(* IEC 61131-3 sources: RL_MAR/experiments/comparison/llm4plc/results/gpt-4o_20260507_114630/20260507_122147, 1 file *)

(* ---- generated_code_iteration_0.st ---- *)
plaintext
START_ST
FUNCTION_BLOCK SoilTestingDeviceControl
VAR_INPUT
    StartButton : BOOL; (* Input for starting the testing process *)
    SoilSampleDetected : BOOL; (* Input for detecting soil sample *)
END_VAR
VAR_OUTPUT
    NutrientPump : BOOL; (* Output to control nutrient pump *)
    pHAdjustmentPump : BOOL; (* Output to control pH adjustment pump *)
END_VAR
VAR
    pHSensorValue : REAL; (* Simulated pH sensor value *)
    NutrientSensorValue : REAL; (* Simulated nutrient sensor value *)
    TestingStatus : INT; (* Status: 0=Idle, 1=Testing, 2=Completed *)
    NutrientThreshold : REAL := 0.7; (* Nutrient level threshold for analysis *)
    pHThreshold : REAL := 6.5; (* pH level threshold for analysis *)
END_VAR

(* Function block logic *)
IF TestingStatus = 0 THEN
    (* STATE 0: Idle *)
    NutrientPump := FALSE;
    pHAdjustmentPump := FALSE;
    pHSensorValue := 7.0; (* Initialize pH sensor value *)
    NutrientSensorValue := 0.5; (* Initialize nutrient sensor value *)

    (* Transition to STATE 1: Testing *)
    IF StartButton THEN
        TestingStatus := 1;
    END_IF;

ELSIF TestingStatus = 1 THEN
    (* STATE 1: Testing *)
    NutrientPump := TRUE;
    pHAdjustmentPump := TRUE;

    (* Simulate sensor value updates *)
    IF NutrientSensorValue < 0.9 THEN
        NutrientSensorValue := NutrientSensorValue + 0.1;
    END_IF;

    IF pHSensorValue > 4.0 THEN
        pHSensorValue := pHSensorValue - 0.5;
    END_IF;

    (* Transition to STATE 2: Completed *)
    IF SoilSampleDetected AND (NutrientSensorValue >= NutrientThreshold) AND (pHSensorValue <= pHThreshold) THEN
        TestingStatus := 2;
    END_IF;

ELSIF TestingStatus = 2 THEN
    (* STATE 2: Completed *)
    NutrientPump := FALSE;
    pHAdjustmentPump := FALSE;

    (* Optionally, add a reset mechanism to transition back to STATE 0 if needed *)
    (* Example:
    IF Reset THEN
        TestingStatus := 0;
    END_IF;
    *)
END_IF;

END_FUNCTION_BLOCK
END_ST
